{attribute 'obsolete' := 'Use E_StatePMPSStatus'}
TYPE ENUM_StatePMPSStatus : E_StatePMPSStatus; END_TYPE

(* stored: Version 1.1.0.1
   DUT ENUM_StatePMPSStatus: Id {b130b5d7-d462-4331-8bc9-7506e97e7cff} *)
